// TwinCAT 3 PLC project Sample
// ProgramVersion: 3.1.4020.2
// libraries:
//   Tc2_Standard, * (Beckhoff Automation GmbH)
//   Tc2_System, * (Beckhoff Automation GmbH)
//   Tc3_Module, * (Beckhoff Automation GmbH)
// project tree:
//   GVLs/ GVL01.TcGVL, GVL02.TcGVL
//   / PlcTask.TcTTO (not stored)
//   POUs/ MAIN.TcPOU

// ---- GVLs/GVL01.TcGVL
{attribute 'qualified_only'}
VAR_GLOBAL
	var01		:	INT;
END_VAR

// ---- GVLs/GVL02.TcGVL
{attribute 'qualified_only'}
VAR_GLOBAL
	var01		:	INT;
END_VAR

// ---- POUs/MAIN.TcPOU
PROGRAM MAIN
VAR
	var01		:	INT;
END_VAR

GVL01.var01 := 1;
GVL02.var01 := 2;
var01 := 3;

END_PROGRAM
